// TIA Portal V16 program export: 5 tag tables, 1 data types, 6 data blocks, 10 code blocks (in call order from the OBs), 3 instance data blocks

VAR_GLOBAL   // PLC tag table "01_Entradas"
   MPistilos_Btn_Start AT %I0.0 : Bool;   // Pulsador Start Pistilos
   MPistilos_Btn_Stop AT %I0.1 : Bool;   // Pulsador Stop Pistilos
   MPistilos_Btn_PE AT %I0.2 : Bool;   // Paro Emergencia Pistilos
   MPistilos_Cam_ST AT %I0.3 : Bool;   // Trigger Pistilos Cam 1
   MPentoflex_Btn_Start AT %I0.4 : Bool;   // Pulsador Start Pentoflex
   MPentoflex_Btn_Stop AT %I0.5 : Bool;   // Pulsador Stop Pentonflex
   MPentoflex_Btn_PE AT %I0.6 : Bool;   // Paro Emergencia Pentoflex
   MPentoflex_Cam_ST AT %I0.7 : Bool;   // Trigger Pentoflex Cam 2
END_VAR

VAR_GLOBAL   // PLC tag table "02_Camara_1"
   "DataMan-TriggerEnable" AT %Q200.0 : Bool;
   "DataMan-Trigger" AT %Q200.1 : Bool;
   "DataMan-TriggerReady" AT %I200.0 : Bool;
   "DataMan-TriggerAck" AT %I200.1 : Bool;
   "DataMan-Acquiring" AT %I200.2 : Bool;
   "DataMan-MissedAcq" AT %I200.3 : Bool;
   "DataMan-TriggerID" AT %IW201 : Word;
   "DataMan-BufferResultsEnable" AT %Q300.0 : Bool;
   "DataMan-ResultsAck" AT %Q300.1 : Bool;
   "DataMan-Decoding" AT %I500.0 : Bool;
   "DataMan-Decode Complete" AT %I500.1 : Bool;
   "DataMan-Results Buffer Overrun" AT %I500.2 : Bool;
   "DataMan-Results Available" AT %I500.3 : Bool;
   "DataMan-General Fault" AT %I500.7 : Bool;
   "DataMan-Train Code" AT %Q600.0 : Bool;
   "DataMan-Train Match String" AT %Q600.1 : Bool;
   "DataMan-Train Focus" AT %Q600.2 : Bool;
   "DataMan-Train Brightness" AT %Q600.3 : Bool;
   "DataMan-Untrain" AT %Q600.4 : Bool;
   "DataMan-Execute DMCC" AT %Q600.6 : Bool;
   "DataMan-Set Match String" AT %Q600.7 : Bool;
   "DataMan-Train Code Ack" AT %I400.0 : Bool;
   "DataMan-Train Match String Ack" AT %I400.1 : Bool;
   "DataMan-Train Focus Ack" AT %I400.2 : Bool;
   "DataMan-Train Brightness Ack" AT %I400.3 : Bool;
   "DataMan-Untrain Ack" AT %I400.4 : Bool;
   "DataMan-Execute DMCC Ack" AT %I400.6 : Bool;
   "DataMan-Set Match String Ack" AT %I400.7 : Bool;
   "DataMan-UserData Option" AT %QW500 : Word;
   "DataMan-UserData Length" AT %QW502 : Word;
   "DataMan-UserData[0]" AT %QB504 : Byte;
   "DataMan-UserData[1]" AT %QB505 : Byte;
   "DataMan-UserData[2]" AT %QB506 : Byte;
   "DataMan-UserData[3]" AT %QB507 : Byte;
   "DataMan-UserData[4]" AT %QB508 : Byte;
   "DataMan-UserData[5]" AT %QB509 : Byte;
   "DataMan-UserData[6]" AT %QB510 : Byte;
   "DataMan-UserData[7]" AT %QB511 : Byte;
   "DataMan-UserData[8]" AT %QB512 : Byte;
   "DataMan-UserData[9]" AT %QB513 : Byte;
   "DataMan-UserData[10]" AT %QB514 : Byte;
   "DataMan-UserData[11]" AT %QB515 : Byte;
   "DataMan-UserData[12]" AT %QB516 : Byte;
   "DataMan-UserData[13]" AT %QB517 : Byte;
   "DataMan-UserData[14]" AT %QB518 : Byte;
   "DataMan-UserData[15]" AT %QB519 : Byte;
   "DataMan-ResultID" AT %IW700 : Word;
   "DataMan-Result Code" AT %IW702 : Word;
   "DataMan-Result Extended" AT %IW704 : Word;
   "DataMan-Result Length" AT %IW706 : Word;
   "DataMan-InspectionResults[0]" AT %IB708 : Byte;
   "DataMan-InspectionResults[1]" AT %IB709 : Byte;
   "DataMan-InspectionResults[2]" AT %IB710 : Byte;
   "DataMan-InspectionResults[3]" AT %IB711 : Byte;
   "DataMan-InspectionResults[4]" AT %IB712 : Byte;
   "DataMan-InspectionResults[5]" AT %IB713 : Byte;
   "DataMan-InspectionResults[6]" AT %IB714 : Byte;
   "DataMan-InspectionResults[7]" AT %IB715 : Byte;
   "DataMan-InspectionResults[8]" AT %IB716 : Byte;
   "DataMan-InspectionResults[9]" AT %IB717 : Byte;
   "DataMan-InspectionResults[10]" AT %IB718 : Byte;
   "DataMan-InspectionResults[11]" AT %IB719 : Byte;
   "DataMan-InspectionResults[12]" AT %IB720 : Byte;
   "DataMan-InspectionResults[13]" AT %IB721 : Byte;
   "DataMan-InspectionResults[14]" AT %IB722 : Byte;
   "DataMan-InspectionResults[15]" AT %IB723 : Byte;
END_VAR

VAR_GLOBAL   // PLC tag table "03_Camara_2"
   "DataMan2-TriggerEnable" AT %Q73.0 : Bool;
   "DataMan2-Trigger" AT %Q73.1 : Bool;
   "DataMan2-TriggerReady" AT %I79.0 : Bool;
   "DataMan2-TriggerAck" AT %I79.1 : Bool;
   "DataMan2-Acquiring" AT %I79.2 : Bool;
   "DataMan2-MissedAcq" AT %I79.3 : Bool;
   "DataMan2-TriggerID" AT %IW80 : Word;
   "DataMan2-BufferResultsEnable" AT %Q74.0 : Bool;
   "DataMan2-ResultsAck" AT %Q74.1 : Bool;
   "DataMan2-Decoding" AT %I82.0 : Bool;
   "DataMan2-Decode Complete" AT %I82.1 : Bool;
   "DataMan2-Results Buffer Overrun" AT %I82.2 : Bool;
   "DataMan2-Results Available" AT %I82.3 : Bool;
   "DataMan2-General Fault" AT %I82.7 : Bool;
   "DataMan2-Train Code" AT %Q75.0 : Bool;
   "DataMan2-Train Match String" AT %Q75.1 : Bool;
   "DataMan2-Train Focus" AT %Q75.2 : Bool;
   "DataMan2-Train Brightness" AT %Q75.3 : Bool;
   "DataMan2-Untrain" AT %Q75.4 : Bool;
   "DataMan2-Execute DMCC" AT %Q75.6 : Bool;
   "DataMan2-Set Match String" AT %Q75.7 : Bool;
   "DataMan2-Train Code Ack" AT %I83.0 : Bool;
   "DataMan2-Train Match String Ack" AT %I83.1 : Bool;
   "DataMan2-Train Focus Ack" AT %I83.2 : Bool;
   "DataMan2-Train Brightness Ack" AT %I83.3 : Bool;
   "DataMan2-Untrain Ack" AT %I83.4 : Bool;
   "DataMan2-Execute DMCC Ack" AT %I83.6 : Bool;
   "DataMan2-Set Match String Ack" AT %I83.7 : Bool;
   "DataMan2-UserData Option" AT %QW76 : Word;
   "DataMan2-UserData Length" AT %QW78 : Word;
   "DataMan2-UserData[0]" AT %QB80 : Byte;
   "DataMan2-UserData[1]" AT %QB81 : Byte;
   "DataMan2-UserData[2]" AT %QB82 : Byte;
   "DataMan2-UserData[3]" AT %QB83 : Byte;
   "DataMan2-UserData[4]" AT %QB84 : Byte;
   "DataMan2-UserData[5]" AT %QB85 : Byte;
   "DataMan2-UserData[6]" AT %QB86 : Byte;
   "DataMan2-UserData[7]" AT %QB87 : Byte;
   "DataMan2-UserData[8]" AT %QB88 : Byte;
   "DataMan2-UserData[9]" AT %QB89 : Byte;
   "DataMan2-UserData[10]" AT %QB90 : Byte;
   "DataMan2-UserData[11]" AT %QB91 : Byte;
   "DataMan2-UserData[12]" AT %QB92 : Byte;
   "DataMan2-UserData[13]" AT %QB93 : Byte;
   "DataMan2-UserData[14]" AT %QB94 : Byte;
   "DataMan2-UserData[15]" AT %QB95 : Byte;
   "DataMan2-ResultID" AT %IW84 : Word;
   "DataMan2-Result Code" AT %IW86 : Word;
   "DataMan2-Result Extended" AT %IW88 : Word;
   "DataMan2-Result Length" AT %IW90 : Word;
   "DataMan2-InspectionResults[0]" AT %IB92 : Byte;
   "DataMan2-InspectionResults[1]" AT %IB93 : Byte;
   "DataMan2-InspectionResults[2]" AT %IB94 : Byte;
   "DataMan2-InspectionResults[3]" AT %IB95 : Byte;
   "DataMan2-InspectionResults[4]" AT %IB96 : Byte;
   "DataMan2-InspectionResults[5]" AT %IB97 : Byte;
   "DataMan2-InspectionResults[6]" AT %IB98 : Byte;
   "DataMan2-InspectionResults[7]" AT %IB99 : Byte;
   "DataMan2-InspectionResults[8]" AT %IB100 : Byte;
   "DataMan2-InspectionResults[9]" AT %IB101 : Byte;
   "DataMan2-InspectionResults[10]" AT %IB102 : Byte;
   "DataMan2-InspectionResults[11]" AT %IB103 : Byte;
   "DataMan2-InspectionResults[12]" AT %IB104 : Byte;
   "DataMan2-InspectionResults[13]" AT %IB105 : Byte;
   "DataMan2-InspectionResults[14]" AT %IB106 : Byte;
   "DataMan2-InspectionResults[15]" AT %IB107 : Byte;
END_VAR

VAR_GLOBAL   // PLC tag table "04_Salidas"
   MPistilos_Motor_Vdf AT %Q0.0 : Bool;   // Motor Pistilos
   MPentoflex_Motor_Logo AT %Q0.1 : Bool;   // Motor Pentoflex
END_VAR

VAR_GLOBAL   // PLC tag table "Tabla de variables estándar"
   System_Byte AT %MB1 : Byte;
   FirstScan AT %M1.0 : Bool;
   DiagStatusUpdate AT %M1.1 : Bool;
   AlwaysTRUE AT %M1.2 : Bool;
   AlwaysFALSE AT %M1.3 : Bool;
   "System_Byte(1)" AT %MB1 : Byte;
   Clock_Byte AT %MB0 : Byte;
   Clock_10Hz AT %M0.0 : Bool;
   Clock_5Hz AT %M0.1 : Bool;
   "Clock_2.5Hz" AT %M0.2 : Bool;
   Clock_2Hz AT %M0.3 : Bool;
   "Clock_1.25Hz" AT %M0.4 : Bool;
   Clock_1Hz AT %M0.5 : Bool;
   "Clock_0.625Hz" AT %M0.6 : Bool;
   "Clock_0.5Hz" AT %M0.7 : Bool;
END_VAR

TYPE "UDT_DatosProd"
// stored: IsFailsafeCompliant false
   STRUCT
      Entradas : Struct
         Longitud : Int;
         Insercion : Bool;
         Dato_In : String;
         Dato_Clr : String;
         Reset : Bool;
         Extraccion : Bool;
      END_STRUCT;
      Salidas : Struct
         Dato_Out : String;
         Add_Dn : Bool;
         Ext_Dn : Bool;
      END_STRUCT;
      Buffer : Array[0..10] of String;
      valor_Camara : String;
   END_STRUCT;
END_TYPE

DATA_BLOCK "01_PLC-Software"   // DB1
{ S7_Optimized_Access := 'TRUE' }
VERSION : 0.1
// stored: AutoNumber true, DBAccessibleFromOPCUA true, IsOnlyStoredInLoadMemory false, IsRetainMemResEnabled false, IsWriteProtectedInAS false, MemoryReserve 100
   VAR
      IN_Pistilos : Array[0..14] of Bool;
      IN_Pentoflex : Array[0..14] of Bool;
      IN_Cam_Pistilos : Array[0..14] of Bool;
      IN_Cam_Pentoflex : Array[0..14] of Bool;
      OUT_Pistilos : Array[0..7] of Bool;
      OUT_Pentoflex : Array[0..7] of Bool;
      Pistilos_Estados_Varidor : Array[0..7] of Bool;
      Alarmas : Array[0..14] of Int;
      Estado_Proceso : Array[0..14] of Bool;
   END_VAR
BEGIN
   // IN_Pistilos[0] : Paro Emerg Pistilos
   // IN_Pistilos[1] : Start Pistilos
   // IN_Pistilos[2] : Stop Pistilos
   // IN_Pistilos[3] : Trigger Cam 1
   // IN_Pentoflex[0] : Paro Emerg Producto Final
   // IN_Pentoflex[1] : Start Producto Final
   // IN_Pentoflex[2] : Stop Producto Final
   // IN_Pentoflex[3] : Trigger Cam 2 Final
   // OUT_Pistilos[0] : Motor Pistilos
   // OUT_Pentoflex[0] : Motor Pentoflex
   // Pistilos_Estados_Varidor[0] : Variador 1 ok
   // Alarmas[0] : Alarma PE Pistilos
   // Alarmas[1] : Alarma_Fallo_Cam_Pistilos
   // Alarmas[2] : Alarma_NLectura_Cam_Pistilos
   // Alarmas[3] : Alarma_NCoincidencia_Cam_Pistilos
   // Alarmas[4] : Alama PE Pentoflex
   // Alarmas[5] : Alarma_Fallo_Cam_Pentoflex
   // Alarmas[6] : Alarma_NLectura_Cam_Pentoflex
   // Alarmas[7] : Alarma_NCoincidencia_Cam_Pentoflex
   // Estado_Proceso[0] : Arranque Modo Automático Pistilos
   // Estado_Proceso[1] : Arranque Modo Manual Pistilos
   // Estado_Proceso[2] : Arranque Modo Automático Pentoflex
   // Estado_Proceso[3] : Arranque Modo Manual Pentoflex
END_DATA_BLOCK

DATA_BLOCK "02_Software-PLC"   // DB2
{ S7_Optimized_Access := 'TRUE' }
VERSION : 0.1
// stored: AutoNumber true, DBAccessibleFromOPCUA true, IsOnlyStoredInLoadMemory false, IsRetainMemResEnabled false, IsWriteProtectedInAS false, MemoryReserve 100
   VAR
      Variables_Generales : Struct
         Multip_Cantiadad_Prod : Real;   // Orden de producción
         Multip_Margen_Prod : Real;   // Margen de error producción
         Multip_Confir_Arranque : Bool;   // Permiso de arranque producción
         Multip_Formato_Trabajo : Int;   // Refencia Cajas
      END_STRUCT;
      Datos_Pentoflex : Struct
         "MPF_Remoto/Local" : Bool;   // Manejo Remoto / Local
         MPF_ModoAuto : Bool;   // Modo Automatico
         MPF_Modo_Manual : Bool;   // Modo Manual
         MPF_Estado_Impresora3 : Bool;   // Estado de la impresora 3
         MPF_Start_Remoto : Bool;   // Start Remoto Pentof
         MPF_Stop_Remoto : Bool;   // Stop Remoto Pentof
         MPF_Reset_Alarmas : Bool;   // Reset Alarma Pentoflex
      END_STRUCT;
      Datos_Pistilos : Struct
         MP_Codigo_Impresion : String;   // codigo de impresión
         MP_Conf_Arranque : Bool;   // Arranque de orden pistilos
         "MP_Remoto/Local" : Bool;   // Manejo Remoto / Local
         MP_ModoAuto : Bool;   // Modo Automatico
         MP_Modo_Manual : Bool;   // Modo Manual
         MP_Estado_Impresora1 : Bool;   // Estado de la impresora 1
         MP_Estado_Impresora2 : Bool;   // Estado de la impresora 2
         MP_Start_Remoto : Bool;   // Start Pistilos Remoto
         MP_Stop_Remoto : Bool;   // Stop Pistilos Remoto
         MP_Cod_Impreso1 : Bool;   // Codigo Impreso
         MP_Reset_Alarmas : Bool;   // Reset Alarmas Pistilos
      END_STRUCT;
   END_VAR
BEGIN
END_DATA_BLOCK

DATA_BLOCK "03_Cam_Pistilos"   // DB3
{ S7_Optimized_Access := 'TRUE' }
VERSION : 0.1
// stored: AutoNumber true, DBAccessibleFromOPCUA true, IsOnlyStoredInLoadMemory false, IsRetainMemResEnabled false, IsWriteProtectedInAS false, MemoryReserve 100
   VAR
      Trigger_Enable_Cam1 : Bool;   // 1= Disparador Ethernet Habilitado
      Trigger : Bool;   // Adquirir imagen
      Status_Register : Array[0..7] of Bool;
      BufferResultsEnable : Bool;
      DecodeStatusRegister : Array[0..7] of Bool;
      ResultsAck : Bool;
      DecodeResult : Struct
         ResultsID : UInt;
         ResultCode : UInt;
         ResultExtended : UInt;
         ResultLength : UInt;
         ResultData : Array[0..63] of Byte;   // Resultados de la ultima decodi
      END_STRUCT;
      SoftEvents : Byte;
      TriggerID : UInt;
      UserDataOption : UInt;
      UserDataLength : UInt;
      SoftEventAck : Byte;
   END_VAR
BEGIN
   Status_Register[0] := true;   // Trigger Ready
   // Status_Register[1] : Trigger Ack
   // Status_Register[2] : Reserved
   // Status_Register[3] : Missed Acquisition
   // Status_Register[4] : Reserved
   // Status_Register[5] : Reserved
   // Status_Register[6] : Reserved
   // Status_Register[7] : Reserved
   // DecodeStatusRegister[0] : Decoding
   // DecodeStatusRegister[1] : Decode Complete
   // DecodeStatusRegister[2] : Result Buffer Overrun
   // DecodeStatusRegister[3] : Result available
   // DecodeStatusRegister[4] : Reserved
   // DecodeStatusRegister[5] : Reserved
   // DecodeStatusRegister[6] : Reserved
   // DecodeStatusRegister[7] : General Fault
END_DATA_BLOCK

DATA_BLOCK "04_Cam_Pentoflex"   // DB4
{ S7_Optimized_Access := 'TRUE' }
VERSION : 0.1
// stored: AutoNumber true, DBAccessibleFromOPCUA true, IsOnlyStoredInLoadMemory false, IsRetainMemResEnabled false, IsWriteProtectedInAS false, MemoryReserve 100
   VAR
      Trigger_Enable_Cam2 : Bool;   // 1= Disparador Ethernet Habilitado
      Trigger : Bool;   // Adquirir imagen
      Status_Register : Array[0..7] of Bool;
      BufferResultsEnable : Bool;
      DecodeStatusRegister : Array[0..7] of Bool;
      ResultsAck : Bool;
      DecodeResult : Struct
         ResultsID : UInt;
         ResultCode : UInt;
         ResultExtended : UInt;
         ResultLength : UInt;
         ResultData : Array[0..63] of Byte;   // Resultados de la ultima decodi
      END_STRUCT;
      SoftEvents : Byte;
      TriggerID : UInt;
      UserDataOption : UInt;
      UserDataLength : UInt;
      SoftEventAck : Byte;
   END_VAR
BEGIN
   Status_Register[0] := true;   // Trigger Ready
   // Status_Register[1] : Trigger Ack
   // Status_Register[2] : Reserved
   // Status_Register[3] : Missed Acquisition
   // Status_Register[4] : Reserved
   // Status_Register[5] : Reserved
   // Status_Register[6] : Reserved
   // Status_Register[7] : Reserved
   // DecodeStatusRegister[0] : Decoding
   // DecodeStatusRegister[1] : Decode Complete
   // DecodeStatusRegister[2] : Result Buffer Overrun
   // DecodeStatusRegister[3] : Result available
   // DecodeStatusRegister[4] : Reserved
   // DecodeStatusRegister[5] : Reserved
   // DecodeStatusRegister[6] : Reserved
   // DecodeStatusRegister[7] : General Fault
END_DATA_BLOCK

DATA_BLOCK "05_General"   // DB5
{ S7_Optimized_Access := 'TRUE' }
VERSION : 0.1
// stored: AutoNumber true, DBAccessibleFromOPCUA true, IsOnlyStoredInLoadMemory false, IsRetainMemResEnabled false, IsWriteProtectedInAS false, MemoryReserve 100
   VAR
      MP_Perifericos_Ok : Bool;   // Confirmación perifericos pistilos
      "MP_Habilita_Start-Stop" : Bool;   // Habilitar Remoto pistilos
      MP_Start_HMI : Bool;   // Start Remoto Pistilos
      MP_Stop_HMI : Bool;   // Stop Remoto Pistilos
      MPF_Perifericos_OK : Bool;   // Confirmación perifericos pentoflex
      "MPF_Habilita_Start-Stop" : Bool;   // Habilitar Remoto pentoflex
      MPF_Start_HMI : Bool;   // Start Remoto Pentoflex
      MP_Stop_HMI_1 : Bool;   // Stop Remoto Pentoflex
   END_VAR
BEGIN
END_DATA_BLOCK

DATA_BLOCK "06_Datos_Produccion"   // DB6
{ S7_Optimized_Access := 'TRUE' }
VERSION : 0.1
// stored: AutoNumber true, DBAccessibleFromOPCUA true, IsOnlyStoredInLoadMemory false, IsRetainMemResEnabled false, IsWriteProtectedInAS false, MemoryReserve 100
   VAR
      Datos_Prod_Pistilos : Struct
         Registro : "UDT_DatosProd";
         Pistilos_ONS : Array[1..10] of Bool;
      END_STRUCT;
      General : Struct
         Indice : Int;
      END_STRUCT;
   END_VAR
BEGIN
   Datos_Prod_Pistilos.Registro.Entradas.Longitud := 10;
END_DATA_BLOCK

ORGANIZATION_BLOCK "Main"   // OB1, LAD, ProgramCycle
TITLE = "Main Program Sweep (Cycle)"
{ S7_Optimized_Access := 'TRUE' }
VERSION : 0.1
// stored: AutoNumber true, IsIECCheckEnabled false, SetENOAutomatically false
   VAR_INPUT
      Initial_Call : Bool;   // Initial call of this OB
      Remanence : Bool;   // =True, if remanent data are available
   END_VAR
   VAR_TEMP   // added for the SCL form of the ladder/FBD networks
      _w1 : Bool;
      _w2 : Bool;
   END_VAR
BEGIN

REGION Network 1
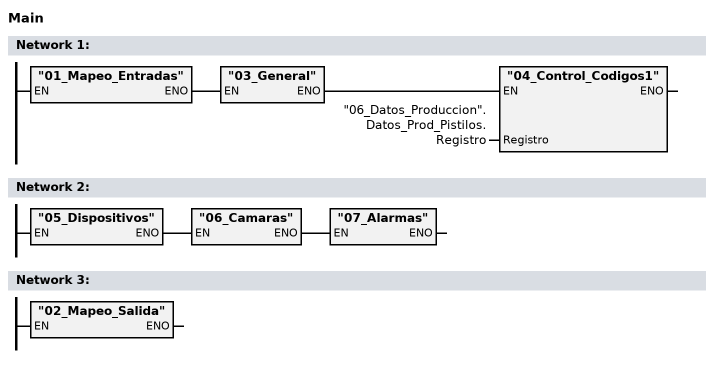
   RUNG wire#powerrail
      "01_Mapeo_Entradas"()
      "03_General"()
      "04_Control_Codigos1"(Registro := "06_Datos_Produccion".Datos_Prod_Pistilos.Registro)
   END_RUNG
   // the same network as SCL:
   "01_Mapeo_Entradas"(ENO => #_w1);
   "03_General"(EN := #_w1, ENO => #_w2);
   IF #_w2 THEN
       "04_Control_Codigos1"(Registro := "06_Datos_Produccion".Datos_Prod_Pistilos.Registro);
   END_IF;
END_REGION

REGION Network 2
   RUNG wire#powerrail
      "05_Dispositivos"()
      "06_Camaras"()
      "07_Alarmas"()
   END_RUNG
   // the same network as SCL:
   "05_Dispositivos"(ENO => #_w1);
   "06_Camaras"(EN := #_w1, ENO => #_w2);
   IF #_w2 THEN "07_Alarmas"(); END_IF;
END_REGION

REGION Network 3
   RUNG wire#powerrail
      "02_Mapeo_Salida"()
   END_RUNG
   // the same network as SCL:
   "02_Mapeo_Salida"();
END_REGION
END_ORGANIZATION_BLOCK

FUNCTION "01_Mapeo_Entradas" : Void   // FC1, LAD
{ S7_Optimized_Access := 'TRUE' }
VERSION : 0.1
// stored: AutoNumber true, IsIECCheckEnabled false, SetENOAutomatically false, UDAEnableTagReadback false
BEGIN

REGION Network 1: Entradas Fisicas Pistilos
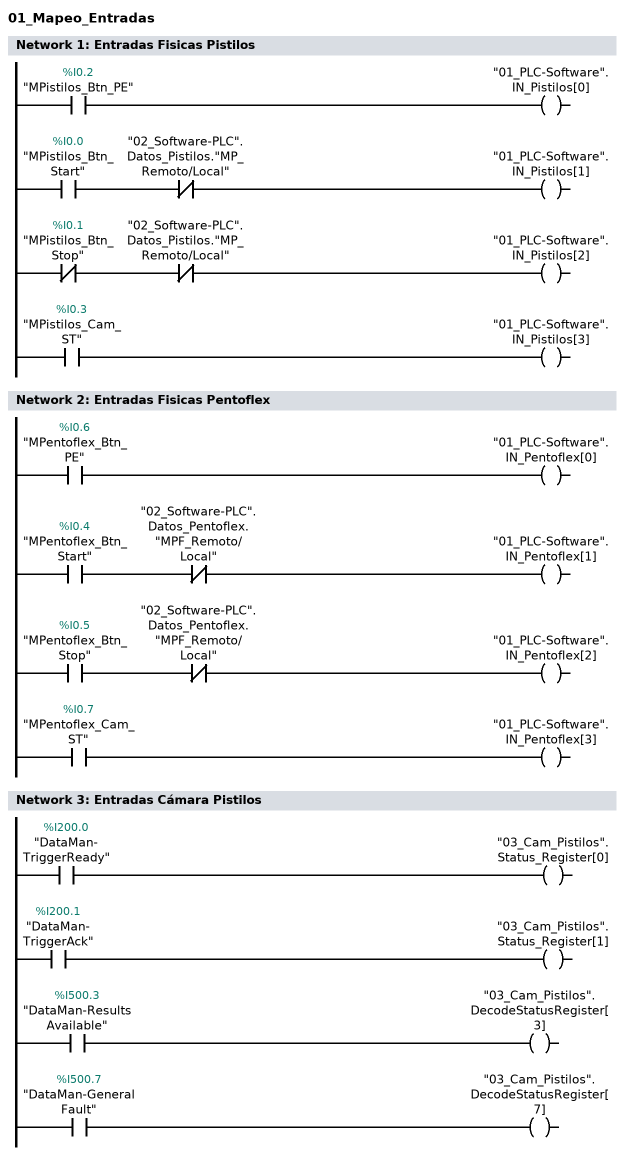
   RUNG wire#powerrail
      Contact( "MPistilos_Btn_PE" )
      Coil( "01_PLC-Software".IN_Pistilos[0] )
   END_RUNG
   RUNG wire#powerrail
      Contact( "MPistilos_Btn_Start" )
      I_Contact( "02_Software-PLC".Datos_Pistilos."MP_Remoto/Local" )
      Coil( "01_PLC-Software".IN_Pistilos[1] )
   END_RUNG
   RUNG wire#powerrail
      I_Contact( "MPistilos_Btn_Stop" )
      I_Contact( "02_Software-PLC".Datos_Pistilos."MP_Remoto/Local" )
      Coil( "01_PLC-Software".IN_Pistilos[2] )
   END_RUNG
   RUNG wire#powerrail
      Contact( "MPistilos_Cam_ST" )
      Coil( "01_PLC-Software".IN_Pistilos[3] )
   END_RUNG
   // the same network as SCL:
   "01_PLC-Software".IN_Pistilos[0] := "MPistilos_Btn_PE";
   "01_PLC-Software".IN_Pistilos[1] := "MPistilos_Btn_Start" AND NOT "02_Software-PLC".Datos_Pistilos."MP_Remoto/Local";
   "01_PLC-Software".IN_Pistilos[2] := NOT "MPistilos_Btn_Stop" AND NOT "02_Software-PLC".Datos_Pistilos."MP_Remoto/Local";
   "01_PLC-Software".IN_Pistilos[3] := "MPistilos_Cam_ST";
END_REGION

REGION Network 2: Entradas Fisicas Pentoflex
   RUNG wire#powerrail
      Contact( "MPentoflex_Btn_PE" )
      Coil( "01_PLC-Software".IN_Pentoflex[0] )
   END_RUNG
   RUNG wire#powerrail
      Contact( "MPentoflex_Btn_Start" )
      I_Contact( "02_Software-PLC".Datos_Pentoflex."MPF_Remoto/Local" )
      Coil( "01_PLC-Software".IN_Pentoflex[1] )
   END_RUNG
   RUNG wire#powerrail
      Contact( "MPentoflex_Btn_Stop" )
      I_Contact( "02_Software-PLC".Datos_Pentoflex."MPF_Remoto/Local" )
      Coil( "01_PLC-Software".IN_Pentoflex[2] )
   END_RUNG
   RUNG wire#powerrail
      Contact( "MPentoflex_Cam_ST" )
      Coil( "01_PLC-Software".IN_Pentoflex[3] )
   END_RUNG
   // the same network as SCL:
   "01_PLC-Software".IN_Pentoflex[0] := "MPentoflex_Btn_PE";
   "01_PLC-Software".IN_Pentoflex[1] := "MPentoflex_Btn_Start" AND NOT "02_Software-PLC".Datos_Pentoflex."MPF_Remoto/Local";
   "01_PLC-Software".IN_Pentoflex[2] := "MPentoflex_Btn_Stop" AND NOT "02_Software-PLC".Datos_Pentoflex."MPF_Remoto/Local";
   "01_PLC-Software".IN_Pentoflex[3] := "MPentoflex_Cam_ST";
END_REGION

REGION Network 3: Entradas Cámara Pistilos
   RUNG wire#powerrail
      Contact( "DataMan-TriggerReady" )
      Coil( "03_Cam_Pistilos".Status_Register[0] )
   END_RUNG
   RUNG wire#powerrail
      Contact( "DataMan-TriggerAck" )
      Coil( "03_Cam_Pistilos".Status_Register[1] )
   END_RUNG
   RUNG wire#powerrail
      Contact( "DataMan-Results Available" )
      Coil( "03_Cam_Pistilos".DecodeStatusRegister[3] )
   END_RUNG
   RUNG wire#powerrail
      Contact( "DataMan-General Fault" )
      Coil( "03_Cam_Pistilos".DecodeStatusRegister[7] )
   END_RUNG
   // the same network as SCL:
   "03_Cam_Pistilos".Status_Register[0] := "DataMan-TriggerReady";
   "03_Cam_Pistilos".Status_Register[1] := "DataMan-TriggerAck";
   "03_Cam_Pistilos".DecodeStatusRegister[3] := "DataMan-Results Available";
   "03_Cam_Pistilos".DecodeStatusRegister[7] := "DataMan-General Fault";
END_REGION

REGION Network 4: Entradas
END_REGION
END_FUNCTION

FUNCTION "03_General" : Void   // FC3, LAD
{ S7_Optimized_Access := 'TRUE' }
VERSION : 0.1
// stored: AutoNumber true, IsIECCheckEnabled false, SetENOAutomatically false, UDAEnableTagReadback false
BEGIN

REGION Network 1: Confirmación Perifericos Pistilos
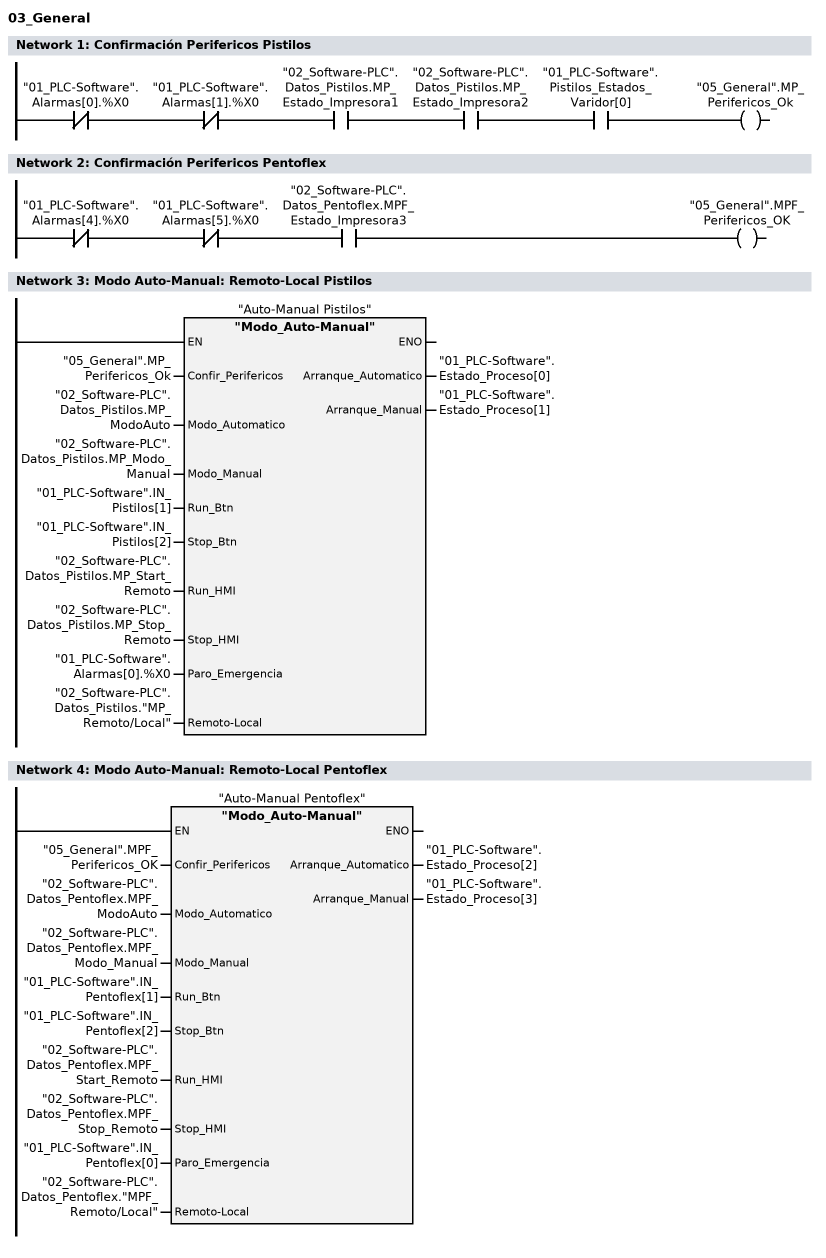
   RUNG wire#powerrail
      I_Contact( "01_PLC-Software".Alarmas[0].%X0 )
      I_Contact( "01_PLC-Software".Alarmas[1].%X0 )
      Contact( "02_Software-PLC".Datos_Pistilos.MP_Estado_Impresora1 )
      Contact( "02_Software-PLC".Datos_Pistilos.MP_Estado_Impresora2 )
      Contact( "01_PLC-Software".Pistilos_Estados_Varidor[0] )
      Coil( "05_General".MP_Perifericos_Ok )
   END_RUNG
   // the same network as SCL:
   "05_General".MP_Perifericos_Ok := NOT "01_PLC-Software".Alarmas[0].%X0 AND NOT "01_PLC-Software".Alarmas[1].%X0 AND "02_Software-PLC".Datos_Pistilos.MP_Estado_Impresora1 AND "02_Software-PLC".Datos_Pistilos.MP_Estado_Impresora2 AND "01_PLC-Software".Pistilos_Estados_Varidor[0];
END_REGION

REGION Network 2: Confirmación Perifericos Pentoflex
   RUNG wire#powerrail
      I_Contact( "01_PLC-Software".Alarmas[4].%X0 )
      I_Contact( "01_PLC-Software".Alarmas[5].%X0 )
      Contact( "02_Software-PLC".Datos_Pentoflex.MPF_Estado_Impresora3 )
      Coil( "05_General".MPF_Perifericos_OK )
   END_RUNG
   // the same network as SCL:
   "05_General".MPF_Perifericos_OK := NOT "01_PLC-Software".Alarmas[4].%X0 AND NOT "01_PLC-Software".Alarmas[5].%X0 AND "02_Software-PLC".Datos_Pentoflex.MPF_Estado_Impresora3;
END_REGION

REGION Network 3: Modo Auto-Manual: Remoto-Local Pistilos
   RUNG wire#powerrail
      "Auto-Manual Pistilos"(Confir_Perifericos := "05_General".MP_Perifericos_Ok, Modo_Automatico := "02_Software-PLC".Datos_Pistilos.MP_ModoAuto, Modo_Manual := "02_Software-PLC".Datos_Pistilos.MP_Modo_Manual, Run_Btn := "01_PLC-Software".IN_Pistilos[1], Stop_Btn := "01_PLC-Software".IN_Pistilos[2], Run_HMI := "02_Software-PLC".Datos_Pistilos.MP_Start_Remoto, Stop_HMI := "02_Software-PLC".Datos_Pistilos.MP_Stop_Remoto, Paro_Emergencia := "01_PLC-Software".Alarmas[0].%X0, "Remoto-Local" := "02_Software-PLC".Datos_Pistilos."MP_Remoto/Local", Arranque_Automatico => "01_PLC-Software".Estado_Proceso[0], Arranque_Manual => "01_PLC-Software".Estado_Proceso[1])
   END_RUNG
   // the same network as SCL:
   "Auto-Manual Pistilos"(Confir_Perifericos := "05_General".MP_Perifericos_Ok,   // "Modo_Auto-Manual"
                          Modo_Automatico := "02_Software-PLC".Datos_Pistilos.MP_ModoAuto,
                          Modo_Manual := "02_Software-PLC".Datos_Pistilos.MP_Modo_Manual,
                          Run_Btn := "01_PLC-Software".IN_Pistilos[1],
                          Stop_Btn := "01_PLC-Software".IN_Pistilos[2],
                          Run_HMI := "02_Software-PLC".Datos_Pistilos.MP_Start_Remoto,
                          Stop_HMI := "02_Software-PLC".Datos_Pistilos.MP_Stop_Remoto,
                          Paro_Emergencia := "01_PLC-Software".Alarmas[0].%X0,
                          "Remoto-Local" := "02_Software-PLC".Datos_Pistilos."MP_Remoto/Local",
                          Arranque_Automatico => "01_PLC-Software".Estado_Proceso[0],
                          Arranque_Manual => "01_PLC-Software".Estado_Proceso[1]);
END_REGION

REGION Network 4: Modo Auto-Manual: Remoto-Local Pentoflex
   RUNG wire#powerrail
      "Auto-Manual Pentoflex"(Confir_Perifericos := "05_General".MPF_Perifericos_OK, Modo_Automatico := "02_Software-PLC".Datos_Pentoflex.MPF_ModoAuto, Modo_Manual := "02_Software-PLC".Datos_Pentoflex.MPF_Modo_Manual, Run_Btn := "01_PLC-Software".IN_Pentoflex[1], Stop_Btn := "01_PLC-Software".IN_Pentoflex[2], Run_HMI := "02_Software-PLC".Datos_Pentoflex.MPF_Start_Remoto, Stop_HMI := "02_Software-PLC".Datos_Pentoflex.MPF_Stop_Remoto, Paro_Emergencia := "01_PLC-Software".IN_Pentoflex[0], "Remoto-Local" := "02_Software-PLC".Datos_Pentoflex."MPF_Remoto/Local", Arranque_Automatico => "01_PLC-Software".Estado_Proceso[2], Arranque_Manual => "01_PLC-Software".Estado_Proceso[3])
   END_RUNG
   // the same network as SCL:
   "Auto-Manual Pentoflex"(Confir_Perifericos := "05_General".MPF_Perifericos_OK,   // "Modo_Auto-Manual"
                           Modo_Automatico := "02_Software-PLC".Datos_Pentoflex.MPF_ModoAuto,
                           Modo_Manual := "02_Software-PLC".Datos_Pentoflex.MPF_Modo_Manual,
                           Run_Btn := "01_PLC-Software".IN_Pentoflex[1],
                           Stop_Btn := "01_PLC-Software".IN_Pentoflex[2],
                           Run_HMI := "02_Software-PLC".Datos_Pentoflex.MPF_Start_Remoto,
                           Stop_HMI := "02_Software-PLC".Datos_Pentoflex.MPF_Stop_Remoto,
                           Paro_Emergencia := "01_PLC-Software".IN_Pentoflex[0],
                           "Remoto-Local" := "02_Software-PLC".Datos_Pentoflex."MPF_Remoto/Local",
                           Arranque_Automatico => "01_PLC-Software".Estado_Proceso[2],
                           Arranque_Manual => "01_PLC-Software".Estado_Proceso[3]);
END_REGION
END_FUNCTION

FUNCTION_BLOCK "Modo_Auto-Manual"   // FB2, LAD
{ S7_Optimized_Access := 'TRUE' }
VERSION : 0.1
// stored: AutoNumber true, IsIECCheckEnabled false, IsRetainMemResEnabled false, MemoryReserve 100, SetENOAutomatically false, UDAEnableTagReadback false
   VAR_INPUT
      Confir_Perifericos : Bool;   // Confirmación Perifericos OK
      Modo_Automatico : Bool;
      Modo_Manual : Bool;
      Run_Btn : Bool;
      Stop_Btn : Bool;
      Run_HMI : Bool;
      Stop_HMI : Bool;
      Paro_Emergencia : Bool;
      "Remoto-Local" : Bool;
   END_VAR
   VAR_OUTPUT
      Arranque_Automatico : Bool;
      Arranque_Manual : Bool;
   END_VAR
   VAR
      Start_Remoto : Bool;
      Stop_Remoto : Bool;
   END_VAR
BEGIN

REGION Network 1: Modo Automático
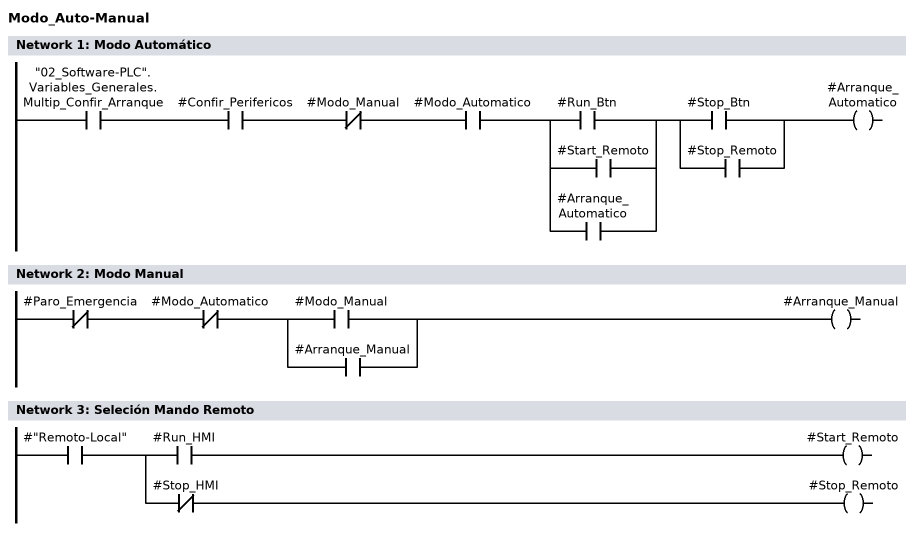
   RUNG wire#powerrail
      Contact( "02_Software-PLC".Variables_Generales.Multip_Confir_Arranque )
      Contact( #Confir_Perifericos )
      I_Contact( #Modo_Manual )
      Contact( #Modo_Automatico )
      wire#w1
      Contact( #Run_Btn )
      wire#w2
      Contact( #Stop_Btn )
      wire#w3
      Coil( #Arranque_Automatico )
   END_RUNG
   RUNG wire#w1
      Contact( #Start_Remoto )
   END_RUNG wire#w2
   RUNG wire#w1
      Contact( #Arranque_Automatico )
   END_RUNG wire#w2
   RUNG wire#w2
      Contact( #Stop_Remoto )
   END_RUNG wire#w3
   // the same network as SCL:
   #Arranque_Automatico := "02_Software-PLC".Variables_Generales.Multip_Confir_Arranque AND #Confir_Perifericos AND NOT #Modo_Manual AND #Modo_Automatico AND (#Run_Btn OR #Start_Remoto OR #Arranque_Automatico) AND (#Stop_Btn OR #Stop_Remoto);
END_REGION

REGION Network 2: Modo Manual
   RUNG wire#powerrail
      I_Contact( #Paro_Emergencia )
      I_Contact( #Modo_Automatico )
      wire#w1
      Contact( #Modo_Manual )
      wire#w2
      Coil( #Arranque_Manual )
   END_RUNG
   RUNG wire#w1
      Contact( #Arranque_Manual )
   END_RUNG wire#w2
   // the same network as SCL:
   #Arranque_Manual := NOT #Paro_Emergencia AND NOT #Modo_Automatico AND (#Modo_Manual OR #Arranque_Manual);
END_REGION

REGION Network 3: Seleción Mando Remoto
   RUNG wire#powerrail
      Contact( #"Remoto-Local" )
      wire#w1
      Contact( #Run_HMI )
      Coil( #Start_Remoto )
   END_RUNG
   RUNG wire#w1
      I_Contact( #Stop_HMI )
      Coil( #Stop_Remoto )
   END_RUNG
   // the same network as SCL:
   #Start_Remoto := #"Remoto-Local" AND #Run_HMI;
   #Stop_Remoto := #"Remoto-Local" AND NOT #Stop_HMI;
END_REGION
END_FUNCTION_BLOCK

FUNCTION "04_Control_Codigos1" : Void   // FC4, LAD
{ S7_Optimized_Access := 'TRUE' }
VERSION : 0.1
// stored: AutoNumber true, IsIECCheckEnabled false, SetENOAutomatically false, UDAEnableTagReadback false
   VAR_IN_OUT
      Registro : "UDT_DatosProd";
   END_VAR
   VAR_TEMP
      i : Int;
      DNC : Bool;
   END_VAR
   VAR_TEMP   // added for the SCL form of the ladder/FBD networks
      _w1 : Bool;
   END_VAR
BEGIN

REGION Network 1
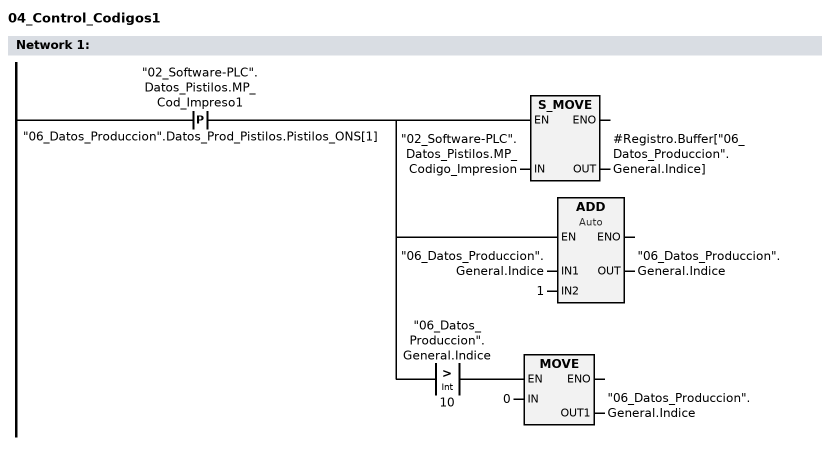
   RUNG wire#powerrail
      P_Contact(operand := "02_Software-PLC".Datos_Pistilos.MP_Cod_Impreso1, bit := "06_Datos_Produccion".Datos_Prod_Pistilos.Pistilos_ONS[1])
      wire#w1
      S_Move(in := "02_Software-PLC".Datos_Pistilos.MP_Codigo_Impresion, out => #Registro.Buffer["06_Datos_Produccion".General.Indice])
   END_RUNG
   RUNG wire#w1
      Add(in1 := "06_Datos_Produccion".General.Indice, in2 := 1, out => "06_Datos_Produccion".General.Indice)
   END_RUNG
   RUNG wire#w1
      { S7_Templates := "SrcType := Int" } GT_Contact(in1 := "06_Datos_Produccion".General.Indice, in2 := 10)
      Move(in := 0, out1 => "06_Datos_Produccion".General.Indice)
   END_RUNG
   // the same network as SCL:
   #_w1 := "02_Software-PLC".Datos_Pistilos.MP_Cod_Impreso1 AND NOT "06_Datos_Produccion".Datos_Prod_Pistilos.Pistilos_ONS[1];   // rising edge of "02_Software-PLC".Datos_Pistilos.MP_Cod_Impreso1
   "06_Datos_Produccion".Datos_Prod_Pistilos.Pistilos_ONS[1] := "02_Software-PLC".Datos_Pistilos.MP_Cod_Impreso1;
   IF #_w1 THEN
       #Registro.Buffer["06_Datos_Produccion".General.Indice] := "02_Software-PLC".Datos_Pistilos.MP_Codigo_Impresion;
       "06_Datos_Produccion".General.Indice := "06_Datos_Produccion".General.Indice + 1;
   END_IF;
   IF #_w1 AND ("06_Datos_Produccion".General.Indice > 10) THEN
       "06_Datos_Produccion".General.Indice := 0;
   END_IF;
END_REGION

REGION Network 3 (SCL)
   IF #Registro.Entradas.Extraccion THEN 
       #Registro.Salidas.Ext_Dn := 1;

       FOR #i := 0 TO #Registro.Entradas.Longitud DO

           IF #Registro.Buffer[#i] = #Registro.valor_Camara THEN

               #Registro.Buffer[#i] := '';
           ELSE
               #DNC := 1;

               EXIT;
           END_IF;

       END_FOR;

   END_IF;
END_REGION
END_FUNCTION

FUNCTION "05_Dispositivos" : Void   // FC5, LAD
{ S7_Optimized_Access := 'TRUE' }
VERSION : 0.1
// stored: AutoNumber true, IsIECCheckEnabled false, SetENOAutomatically false, UDAEnableTagReadback false
BEGIN
END_FUNCTION

FUNCTION "06_Camaras" : Void   // FC6, LAD
{ S7_Optimized_Access := 'TRUE' }
VERSION : 0.1
// stored: AutoNumber true, IsIECCheckEnabled false, SetENOAutomatically false, UDAEnableTagReadback false
BEGIN

REGION Network 1: Bloque Cámara Pistilos
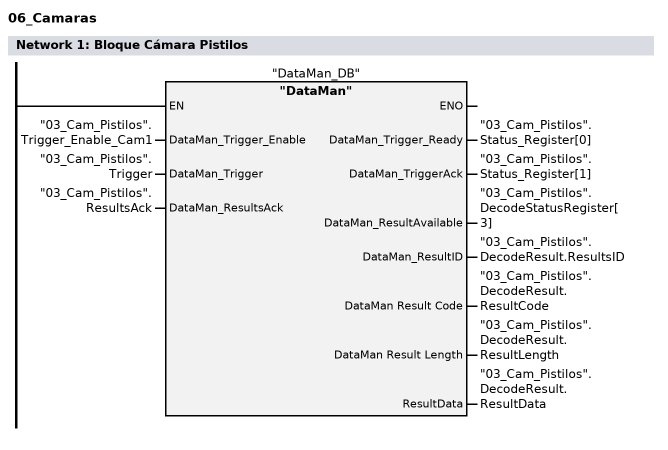
   RUNG wire#powerrail
      "DataMan_DB"(DataMan_Trigger_Enable := "03_Cam_Pistilos".Trigger_Enable_Cam1, DataMan_Trigger := "03_Cam_Pistilos".Trigger, DataMan_ResultsAck := "03_Cam_Pistilos".ResultsAck, DataMan_Trigger_Ready => "03_Cam_Pistilos".Status_Register[0], DataMan_TriggerAck => "03_Cam_Pistilos".Status_Register[1], DataMan_ResultAvailable => "03_Cam_Pistilos".DecodeStatusRegister[3], DataMan_ResultID => "03_Cam_Pistilos".DecodeResult.ResultsID, "DataMan Result Code" => "03_Cam_Pistilos".DecodeResult.ResultCode, "DataMan Result Length" => "03_Cam_Pistilos".DecodeResult.ResultLength, ResultData => "03_Cam_Pistilos".DecodeResult.ResultData)
   END_RUNG
   // the same network as SCL:
   "DataMan_DB"(DataMan_Trigger_Enable := "03_Cam_Pistilos".Trigger_Enable_Cam1,   // "DataMan"
                DataMan_Trigger := "03_Cam_Pistilos".Trigger,
                DataMan_ResultsAck := "03_Cam_Pistilos".ResultsAck,
                DataMan_Trigger_Ready => "03_Cam_Pistilos".Status_Register[0],
                DataMan_TriggerAck => "03_Cam_Pistilos".Status_Register[1],
                DataMan_ResultAvailable => "03_Cam_Pistilos".DecodeStatusRegister[3],
                DataMan_ResultID => "03_Cam_Pistilos".DecodeResult.ResultsID,
                "DataMan Result Code" => "03_Cam_Pistilos".DecodeResult.ResultCode,
                "DataMan Result Length" => "03_Cam_Pistilos".DecodeResult.ResultLength,
                ResultData => "03_Cam_Pistilos".DecodeResult.ResultData);
END_REGION
END_FUNCTION

FUNCTION_BLOCK "DataMan"   // FB1, LAD
TITLE = Cámara Cognex DataMan
{ S7_Optimized_Access := 'TRUE' }
VERSION : 0.1
// stored: AutoNumber true, IsIECCheckEnabled false, IsRetainMemResEnabled false, MemoryReserve 100, SetENOAutomatically false, UDAEnableTagReadback false
   VAR_OUTPUT
      DataMan_Trigger_Ready : Bool;
      DataMan_TriggerAck : Bool;
      DataMan_ResultAvailable : Bool;
      DataMan_ResultID : Word;
      "DataMan Result Code" : Word;
      "DataMan Result Length" : Word;
      ResultData : Array[0..63] of Byte;
   END_VAR
   VAR_IN_OUT
      DataMan_Trigger_Enable : Bool;
      DataMan_Trigger : Bool;
      DataMan_ResultsAck : Bool;
   END_VAR
   VAR
      Resultado_Pendiente : Bool;
      "Lastest Result" : Struct
         ID : Int;
         Flags : Int;
         Lenght : Int;
         Value : Array[0..63] of Byte;
      END_STRUCT;
   END_VAR
   VAR_TEMP   // added for the SCL form of the ladder/FBD networks
      _w1 : Bool;
   END_VAR
BEGIN

REGION Network 1: Habilitar Comunicación Profinet
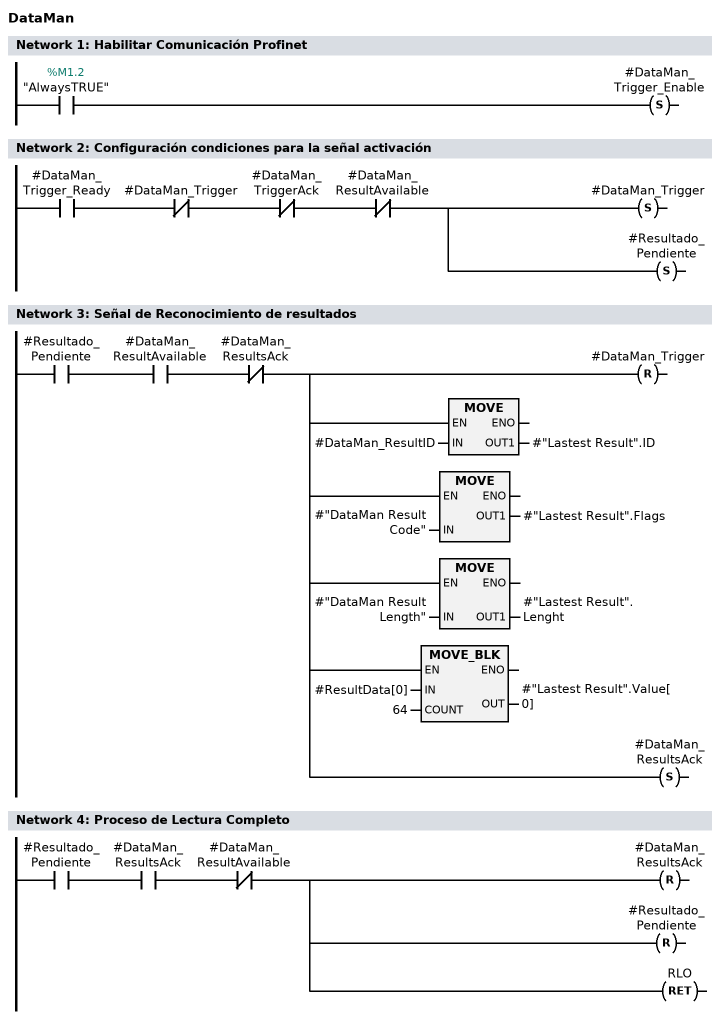
   RUNG wire#powerrail
      Contact( "AlwaysTRUE" )
      S_Coil( #DataMan_Trigger_Enable )
   END_RUNG
   // the same network as SCL:
   IF "AlwaysTRUE" THEN #DataMan_Trigger_Enable := TRUE; END_IF;
END_REGION

REGION Network 2: Configuración condiciones para la señal activación
   RUNG wire#powerrail
      Contact( #DataMan_Trigger_Ready )
      I_Contact( #DataMan_Trigger )
      I_Contact( #DataMan_TriggerAck )
      I_Contact( #DataMan_ResultAvailable )
      wire#w1
      S_Coil( #DataMan_Trigger )
   END_RUNG
   RUNG wire#w1
      S_Coil( #Resultado_Pendiente )
   END_RUNG
   // the same network as SCL:
   #_w1 := #DataMan_Trigger_Ready AND NOT #DataMan_Trigger AND NOT #DataMan_TriggerAck AND NOT #DataMan_ResultAvailable;
   IF #_w1 THEN
       #DataMan_Trigger := TRUE;
       #Resultado_Pendiente := TRUE;
   END_IF;
END_REGION

REGION Network 3: Señal de Reconocimiento de resultados
   IF #Resultado_Pendiente AND #DataMan_ResultAvailable AND NOT #DataMan_ResultsAck THEN
       #DataMan_Trigger := FALSE;
       #"Lastest Result".ID := #DataMan_ResultID;
       #"Lastest Result".Flags := #"DataMan Result Code";
       #"Lastest Result".Lenght := #"DataMan Result Length";
       MOVE_BLK(IN := #ResultData[0], COUNT := 64, OUT => #"Lastest Result".Value[0]);
       #DataMan_ResultsAck := TRUE;
   END_IF;
END_REGION

REGION Network 4: Proceso de Lectura Completo
   #_w1 := #Resultado_Pendiente AND #DataMan_ResultsAck AND NOT #DataMan_ResultAvailable;
   IF #_w1 THEN
       #DataMan_ResultsAck := FALSE;
       #Resultado_Pendiente := FALSE;
       ENO := TRUE;
       RETURN;
   END_IF;
END_REGION
END_FUNCTION_BLOCK

FUNCTION "07_Alarmas" : Void   // FC7, LAD
TITLE = Alarmas
{ S7_Optimized_Access := 'TRUE' }
VERSION : 0.1
// stored: AutoNumber true, IsIECCheckEnabled false, SetENOAutomatically false, UDAEnableTagReadback false
BEGIN

REGION Network 1: Paro Emergencia Pistilos
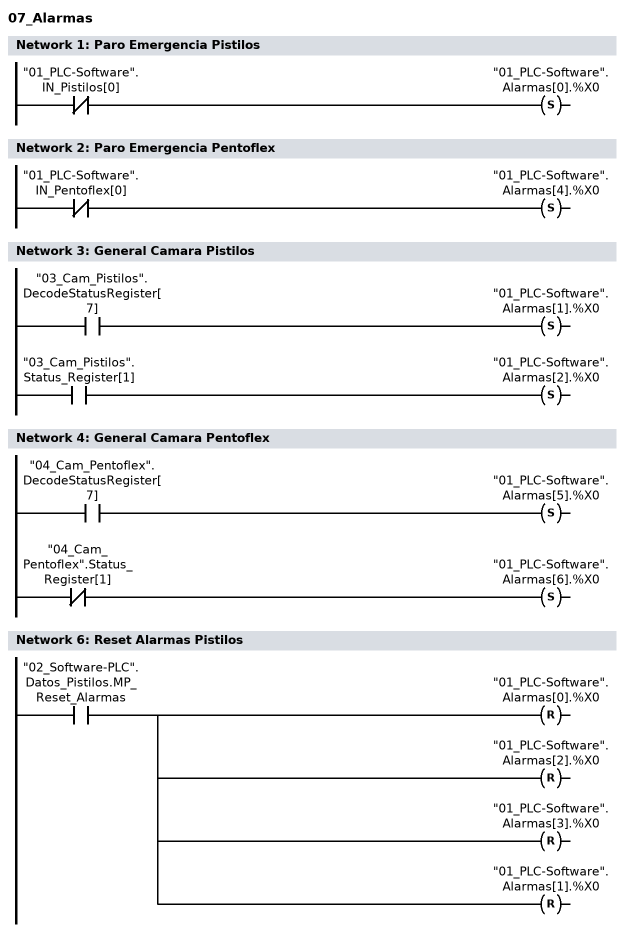
   RUNG wire#powerrail
      I_Contact( "01_PLC-Software".IN_Pistilos[0] )
      S_Coil( "01_PLC-Software".Alarmas[0].%X0 )
   END_RUNG
   // the same network as SCL:
   IF NOT "01_PLC-Software".IN_Pistilos[0] THEN "01_PLC-Software".Alarmas[0].%X0 := TRUE; END_IF;
END_REGION

REGION Network 2: Paro Emergencia Pentoflex
   RUNG wire#powerrail
      I_Contact( "01_PLC-Software".IN_Pentoflex[0] )
      S_Coil( "01_PLC-Software".Alarmas[4].%X0 )
   END_RUNG
   // the same network as SCL:
   IF NOT "01_PLC-Software".IN_Pentoflex[0] THEN "01_PLC-Software".Alarmas[4].%X0 := TRUE; END_IF;
END_REGION

REGION Network 3: General Camara Pistilos
   RUNG wire#powerrail
      Contact( "03_Cam_Pistilos".DecodeStatusRegister[7] )
      S_Coil( "01_PLC-Software".Alarmas[1].%X0 )
   END_RUNG
   RUNG wire#powerrail
      Contact( "03_Cam_Pistilos".Status_Register[1] )
      S_Coil( "01_PLC-Software".Alarmas[2].%X0 )
   END_RUNG
   // the same network as SCL:
   IF "03_Cam_Pistilos".DecodeStatusRegister[7] THEN "01_PLC-Software".Alarmas[1].%X0 := TRUE; END_IF;
   IF "03_Cam_Pistilos".Status_Register[1] THEN "01_PLC-Software".Alarmas[2].%X0 := TRUE; END_IF;
END_REGION

REGION Network 4: General Camara Pentoflex
   RUNG wire#powerrail
      Contact( "04_Cam_Pentoflex".DecodeStatusRegister[7] )
      S_Coil( "01_PLC-Software".Alarmas[5].%X0 )
   END_RUNG
   RUNG wire#powerrail
      I_Contact( "04_Cam_Pentoflex".Status_Register[1] )
      S_Coil( "01_PLC-Software".Alarmas[6].%X0 )
   END_RUNG
   // the same network as SCL:
   IF "04_Cam_Pentoflex".DecodeStatusRegister[7] THEN "01_PLC-Software".Alarmas[5].%X0 := TRUE; END_IF;
   IF NOT "04_Cam_Pentoflex".Status_Register[1] THEN "01_PLC-Software".Alarmas[6].%X0 := TRUE; END_IF;
END_REGION

REGION Network 5: Variador
END_REGION

REGION Network 6: Reset Alarmas Pistilos
   RUNG wire#powerrail
      Contact( "02_Software-PLC".Datos_Pistilos.MP_Reset_Alarmas )
      wire#w1
      R_Coil( "01_PLC-Software".Alarmas[0].%X0 )
   END_RUNG
   RUNG wire#w1
      R_Coil( "01_PLC-Software".Alarmas[2].%X0 )
   END_RUNG
   RUNG wire#w1
      R_Coil( "01_PLC-Software".Alarmas[3].%X0 )
   END_RUNG
   RUNG wire#w1
      R_Coil( "01_PLC-Software".Alarmas[1].%X0 )
   END_RUNG
   // the same network as SCL:
   IF "02_Software-PLC".Datos_Pistilos.MP_Reset_Alarmas THEN
       "01_PLC-Software".Alarmas[0].%X0 := FALSE;
       "01_PLC-Software".Alarmas[2].%X0 := FALSE;
       "01_PLC-Software".Alarmas[3].%X0 := FALSE;
       "01_PLC-Software".Alarmas[1].%X0 := FALSE;
   END_IF;
END_REGION
END_FUNCTION

FUNCTION "02_Mapeo_Salida" : Void   // FC2, LAD
{ S7_Optimized_Access := 'TRUE' }
VERSION : 0.1
// stored: AutoNumber true, IsIECCheckEnabled false, SetENOAutomatically false, UDAEnableTagReadback false
BEGIN

REGION Network 1: Salidas Pistilos
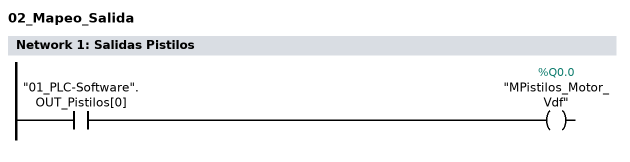
   RUNG wire#powerrail
      Contact( "01_PLC-Software".OUT_Pistilos[0] )
      Coil( "MPistilos_Motor_Vdf" )
   END_RUNG
   // the same network as SCL:
   "MPistilos_Motor_Vdf" := "01_PLC-Software".OUT_Pistilos[0];
END_REGION
END_FUNCTION

DATA_BLOCK "Auto-Manual Pentoflex"   // DB8
VERSION : 0.1
// stored: AutoNumber true, DBAccessibleFromOPCUA true, InstanceOfName Modo_Auto-Manual, InstanceOfType FB
"Modo_Auto-Manual"
BEGIN
END_DATA_BLOCK

DATA_BLOCK "Auto-Manual Pistilos"   // DB7
VERSION : 0.1
// stored: AutoNumber true, DBAccessibleFromOPCUA true, InstanceOfName Modo_Auto-Manual, InstanceOfType FB
"Modo_Auto-Manual"
BEGIN
END_DATA_BLOCK

DATA_BLOCK "DataMan_DB"   // DB9
VERSION : 0.1
// stored: AutoNumber true, DBAccessibleFromOPCUA true, InstanceOfName DataMan, InstanceOfType FB
"DataMan"
BEGIN
END_DATA_BLOCK
